FUNCTION_BLOCK READER2
  {SET_ATTRIBUTE(OpcUa, SERVICE)}
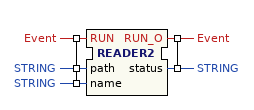
  EVENT_INPUT
    RUN WITH path, name; {SET_ATTRIBUTE(OpcUa, Method)}
  END_EVENT
  EVENT_OUTPUT
    RUN_O WITH status;
  END_EVENT
  VAR_INPUT
    path : STRING; {SET_ATTRIBUTE(OpcUa, Variable.RUN)}
    name : STRING; {SET_ATTRIBUTE(OpcUa, Variable.RUN)}
  END_VAR
  VAR_OUTPUT
    status : STRING; {SET_ATTRIBUTE(OpcUa, Variable.RUN)}
  END_VAR
END_FUNCTION_BLOCK
